FUNCTION_BLOCK PRINT (* Prints a value or vector on the screen *)
  (* Standard: 61499-2 *)
  (* Version 1.0, 01-06-12, GASR, Universidade do Estado de Santa Catarina *)
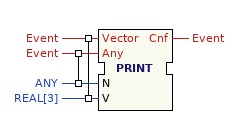
  EVENT_INPUT
    Vector WITH V;
    Any WITH N;
  END_EVENT
  EVENT_OUTPUT
    Cnf;
  END_EVENT
  VAR_INPUT
    N : ANY;
    V : ARRAY [0..2] OF REAL;
  END_VAR
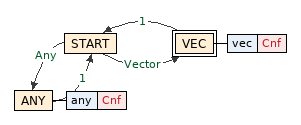
  EC_STATES
    VEC : vec -> Cnf;
    START;
    ANY : any -> Cnf;
  END_STATES
  EC_TRANSITIONS
    START TO VEC := Vector;
    START TO ANY := Any;
    VEC TO START := 1;
    ANY TO START := 1;
  END_TRANSITIONS
  ALGORITHM vec IN Lua:
 print( 'Print FB', V[1], V[2], V[3] )
  END_ALGORITHM
  ALGORITHM any IN Lua:
 print( 'Print FB', N )
  END_ALGORITHM
END_FUNCTION_BLOCK
